{attribute 'qualified_only'}
{attribute 'to_string'}
TYPE eFeed :
(
	Stop := 0,
	Ready,
	Running,
	Fault,
	State4
);
END_TYPE

(* stored: Version 1.1.0.1, ProductVersion 3.1.4024.10
   DUT eFeed: Id {f55bf0d3-82f8-4b9d-a937-5772250db59f} *)
